TYPE EL6002_COM_Inputs :
STRUCT
	{attribute addProperty Name "Status"}
	Status AT %I* : EL6002_Status;
	{attribute addProperty Name "Data"}
	Data  AT %I* : ARRAY[0..21] OF USINT;
END_STRUCT
END_TYPE

(* stored: Version 1.1.0.1, ProductVersion 3.1.4024.9
   DUT EL6002_COM_Inputs: Id {a2d5586a-0848-0306-2a4e-3e7acd7ff7fd} *)
